Staubli VAL3: Safety.pgx

program Safety()
begin
  do

    // Rearme del safety
    if diSafetyRearme==true and esStatus()==1
      setSafetyRestart()
    endIf


  until false
end
